// TIA Portal V17 export
// export: Created 2022-03-12T16:05:35.480794Z, ExportSetting WithDefaults, DisplayName Totally Integrated Automation Portal, DisplayVersion V17, DisplayName TIA Portal Openness, DisplayVersion V17, DisplayName TIA Portal Version Control Interface, DisplayVersion V17, DisplayName STEP 7 Professional, DisplayVersion V17, DisplayName STEP 7 Safety, DisplayVersion V17, DisplayName WinCC Advanced / Unified PC, DisplayVersion V17
TYPE "typeLPMLV30_DiagnosticsEntry"
TITLE = typeLPMLV30_DiagnosticsEntry
// Support: tech.team.motioncontrol@siemens.com 
// Fax: +49 (0) 9131/98-1297
// stored: IsFailsafeCompliant false
   STRUCT
      timestamp : DTL := DTL#1970-01-01-00:00:00;   // Timestamp for this entry
      UnitModeCurrent : Byte := 16#00;   // Current unit mode
      StateCurrent : Byte := 16#00;   // Current state
      UnitMode : Byte := 16#00;   // Requested unit mode
      CntrlCmd : Byte := 16#00;   // Request control command
      SC : Bool := false;   // State complete signal
      message : Byte := 16#00;   // Message for this entry
   END_STRUCT;
END_TYPE
